FUNCTION_BLOCK PUBLIC FB_Publisher IMPLEMENTS I_Publisher
VAR	
	fbDelay				: TON;
	fbDrand				: DRAND;
	_Value				: LREAL;
	aSubscribers		: ARRAY [1..Param.MaxSubscribers] OF I_Subscriber;
END_VAR

// creates every sec a random value and invoke the update method
fbDelay(IN := TRUE, PT := T#1S);
IF (fbDelay.Q) THEN	
	fbDelay(IN := FALSE);	
	fbDrand(SEED := 0);
	_Value := fbDrand.Num * 1234.5;
	NotifySubscribers();
END_IF

PROPERTY ActualValue : LREAL
GET
ActualValue := THIS^._Value;
END_GET
END_PROPERTY

METHOD PUBLIC AddSubscriber : BOOL
VAR_INPUT
	ipSubscriber	: I_Subscriber;
END_VAR
VAR
	nIndex					: INT := 0;
END_VAR
AddSubscriber := FALSE;
IF (ipSubscriber = 0) THEN
	RETURN;
END_IF

// is the observer already registered?
FOR nIndex := 1 TO Param.MaxSubscribers DO	
	IF (THIS^.aSubscribers[nIndex] = ipSubscriber) THEN
		RETURN;
	END_IF
END_FOR

// save the observer object into the array of observers and send the actual value
FOR nIndex := 1 TO Param.MaxSubscribers DO
	IF (THIS^.aSubscribers[nIndex] = 0) THEN
		THIS^.aSubscribers[nIndex] := ipSubscriber;
		THIS^.aSubscribers[nIndex].Update(THIS^._Value);
		AddSubscriber := TRUE;
		EXIT;					
	END_IF
END_FOR
END_METHOD

METHOD PRIVATE NotifySubscribers : BOOL
VAR	
	nIndex	: INT := 0;
END_VAR
FOR nIndex := 1 TO Param.MaxSubscribers DO
	IF (THIS^.aSubscribers[nIndex] <> 0) THEN
		THIS^.aSubscribers[nIndex].Update(THIS^.ActualValue);
	END_IF
END_FOR
END_METHOD

METHOD RemoveSubscriber : BOOL
VAR_INPUT
	ipSubscriber	: I_Subscriber;
END_VAR
VAR
	nIndex			: INT := 0;
END_VAR
RemoveSubscriber := FALSE;
IF (ipSubscriber = 0) THEN
	RETURN;
END_IF

FOR nIndex := 1 TO Param.MaxSubscribers DO
	IF (THIS^.aSubscribers[nIndex] = ipSubscriber) THEN
		THIS^.aSubscribers[nIndex] := 0;
		RemoveSubscriber := TRUE;	
	END_IF
END_FOR
END_METHOD

END_FUNCTION_BLOCK

(* stored: Version 1.1.0.1, ProductVersion 3.1.4022.18
   POU FB_Publisher: Id {ca1a5934-51b6-43f8-b9d0-3eecb1e2da99}, SpecialFunc None
   Property ActualValue: Id {965a95ab-3222-4556-b092-10eca8d71ba5}
   Get Get: Id {bce8c020-8c39-40fc-9ec9-bb7942710e4d}
   Method AddSubscriber: Id {f0060a5f-66e9-47a2-82f9-d9a36c2a08e9}
   Method NotifySubscribers: Id {dac65567-2911-4040-aa40-37d939ba993a}
   Method RemoveSubscriber: Id {813c32e8-adda-40cf-b613-8bd62e562b69} *)
